TYPE ST_PowerModule_calibration :
STRUCT
	b_StartCalibration			: BOOL;
	r_Pset						: REAL;
	r_Qset						: REAL;
	PCoefficients				: ST_Powermodule_PowerCurveCoefficients;
	QCoefficients				: ST_Powermodule_PowerCurveCoefficients;
	CalibrationData				: ST_Powermodule_calibData;
END_STRUCT
END_TYPE

(* stored: Version 1.1.0.1, ProductVersion 3.1.4026.18
   DUT ST_PowerModule_calibration: Id {354e619d-0332-45bc-833e-e692cf370a9a} *)
